FUNCTION_BLOCK E_F_TRIG
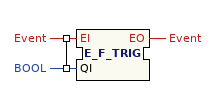
  EVENT_INPUT
    EI WITH QI;
  END_EVENT
  EVENT_OUTPUT
    EO;
  END_EVENT
  VAR_INPUT
    QI : BOOL;
  END_VAR
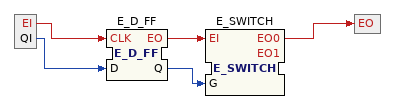
  FBS
    E_D_FF : E_D_FF;
    E_SWITCH : E_SWITCH;
  END_FBS
  EVENT_CONNECTIONS
    EI TO E_D_FF.CLK;
    E_D_FF.EO TO E_SWITCH.EI;
    E_SWITCH.EO0 TO EO;
  END_CONNECTIONS
  DATA_CONNECTIONS
    QI TO E_D_FF.D;
    E_D_FF.Q TO E_SWITCH.G;
  END_CONNECTIONS
END_FUNCTION_BLOCK
